// TIA Portal V17 export
// export: Created 2023-05-12T10:40:25.6107869Z, DisplayName Totally Integrated Automation Portal, DisplayVersion V17 Update 4, DisplayName TIA Portal Openness, DisplayVersion V17 Update 4, DisplayName TIA Portal Version Control Interface, DisplayVersion V17, DisplayName STEP 7 Professional, DisplayVersion V17 Update 4, DisplayName STEP 7 Safety, DisplayVersion V17, DisplayName WinCC Advanced / Unified PC, DisplayVersion V17 Update 4
FUNCTION_BLOCK "FB_EM_InputConditioning"   // FB19, LAD
{ S7_Optimized_Access := 'TRUE' }
VERSION : 0.1
// stored: AutoNumber true, CodeModifiedDate 2023-05-12T12:59:41.6492354Z, CompileDate 2023-05-12T12:59:41.6492354Z, CreationDate 2023-05-08T12:19:11.3376827Z, DownloadWithoutReinit false, HandleErrorsWithinBlock false, InterfaceModifiedDate 2023-05-12T12:59:19.7337351Z, IsConsistent true, IsIECCheckEnabled false, IsKnowHowProtected false, IsRetainMemResEnabled false, IsWriteProtected false, LibraryConformanceStatus Warning: The object contains access to global data blocks., MemoryReserve 100, ModifiedDate 2023-05-12T12:59:41.6492354Z, ParameterModified 2022-09-13T10:25:33.4387708Z, PLCSimAdvancedSupport true, SetENOAutomatically false, StructureModified 2023-05-12T12:59:19.7337351Z, UDAEnableTagReadback false
   VAR
      FT01_Przeplyw_Inst { S7_SetPoint := 'True'} : "FB_CM_MeasurementPoint";
      TTs_TempSzafy_Inst { S7_SetPoint := 'True'} : "FB_CM_MeasurementPoint";
      TTz_TempZewn_Inst { S7_SetPoint := 'True'} : "FB_CM_MeasurementPoint";
      PT07_CisnZasil_WRZ6_Inst { S7_SetPoint := 'True'} : "FB_CM_MeasurementPoint";
      PT08_CisnPowr_WRZ6_Inst { S7_SetPoint := 'True'} : "FB_CM_MeasurementPoint";
      TTk_TempKom_Inst { S7_SetPoint := 'True'} : "FB_CM_MeasurementPoint";
      PT01_CisnZasil_PLN1_Inst { S7_SetPoint := 'True'} : "FB_CM_MeasurementPoint";
      PT02_CisnPowr_PLN1_Inst { S7_SetPoint := 'True'} : "FB_CM_MeasurementPoint";
      PT03_CisnZasil_Bypass_Inst { S7_SetPoint := 'True'} : "FB_CM_MeasurementPoint";
      PT04_CisnPowr_Bypass_Inst { S7_SetPoint := 'True'} : "FB_CM_MeasurementPoint";
      PT05_CisnZasil_PLN12_Inst { S7_SetPoint := 'True'} : "FB_CM_MeasurementPoint";
      PT06_CisnPowr_PLN12_Inst { S7_SetPoint := 'True'} : "FB_CM_MeasurementPoint";
      TT01_TempZasil_PLN1_Inst { S7_SetPoint := 'True'} : "FB_CM_MeasurementPoint";
      TT02_TempPowr_PLN1_Inst { S7_SetPoint := 'True'} : "FB_CM_MeasurementPoint";
      TT04_TempPowr_WRZ6_Inst { S7_SetPoint := 'True'} : "FB_CM_MeasurementPoint";
      TT06_TempPowr_PLN12_Inst { S7_SetPoint := 'True'} : "FB_CM_MeasurementPoint";
   END_VAR
BEGIN

REGION Network 1: FT01_Przeplyw - Przepływ
   // FT01_Przeplyw - Przepływ
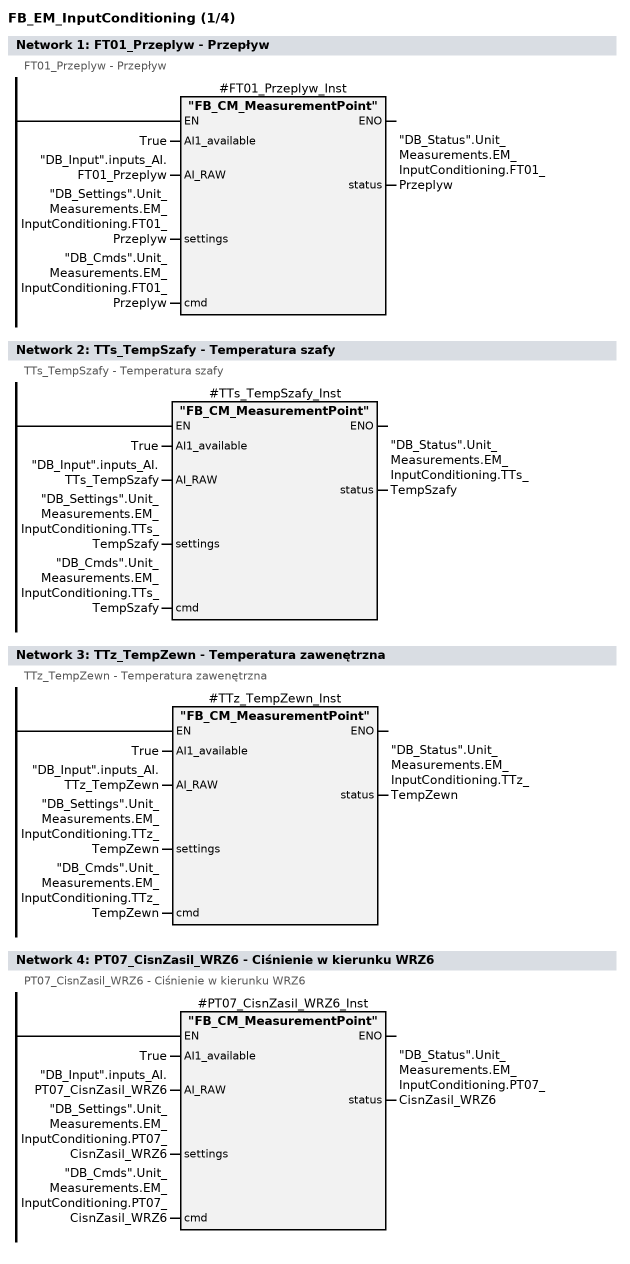
   RUNG wire#powerrail
      #FT01_Przeplyw_Inst(AI1_available := True, AI_RAW := "DB_Input".inputs_AI.FT01_Przeplyw, settings := "DB_Settings".Unit_Measurements.EM_InputConditioning.FT01_Przeplyw, cmd := "DB_Cmds".Unit_Measurements.EM_InputConditioning.FT01_Przeplyw, status => "DB_Status".Unit_Measurements.EM_InputConditioning.FT01_Przeplyw)
   END_RUNG
   // the same network as SCL:
   #FT01_Przeplyw_Inst(AI1_available := True,   // "FB_CM_MeasurementPoint"
                       AI_RAW := "DB_Input".inputs_AI.FT01_Przeplyw,
                       settings := "DB_Settings".Unit_Measurements.EM_InputConditioning.FT01_Przeplyw,
                       cmd := "DB_Cmds".Unit_Measurements.EM_InputConditioning.FT01_Przeplyw,
                       status => "DB_Status".Unit_Measurements.EM_InputConditioning.FT01_Przeplyw);
END_REGION

REGION Network 2: TTs_TempSzafy - Temperatura szafy
   // TTs_TempSzafy - Temperatura szafy
   RUNG wire#powerrail
      #TTs_TempSzafy_Inst(AI1_available := True, AI_RAW := "DB_Input".inputs_AI.TTs_TempSzafy, settings := "DB_Settings".Unit_Measurements.EM_InputConditioning.TTs_TempSzafy, cmd := "DB_Cmds".Unit_Measurements.EM_InputConditioning.TTs_TempSzafy, status => "DB_Status".Unit_Measurements.EM_InputConditioning.TTs_TempSzafy)
   END_RUNG
   // the same network as SCL:
   #TTs_TempSzafy_Inst(AI1_available := True,   // "FB_CM_MeasurementPoint"
                       AI_RAW := "DB_Input".inputs_AI.TTs_TempSzafy,
                       settings := "DB_Settings".Unit_Measurements.EM_InputConditioning.TTs_TempSzafy,
                       cmd := "DB_Cmds".Unit_Measurements.EM_InputConditioning.TTs_TempSzafy,
                       status => "DB_Status".Unit_Measurements.EM_InputConditioning.TTs_TempSzafy);
END_REGION

REGION Network 3: TTz_TempZewn - Temperatura zawenętrzna
   // TTz_TempZewn - Temperatura zawenętrzna
   RUNG wire#powerrail
      #TTz_TempZewn_Inst(AI1_available := True, AI_RAW := "DB_Input".inputs_AI.TTz_TempZewn, settings := "DB_Settings".Unit_Measurements.EM_InputConditioning.TTz_TempZewn, cmd := "DB_Cmds".Unit_Measurements.EM_InputConditioning.TTz_TempZewn, status => "DB_Status".Unit_Measurements.EM_InputConditioning.TTz_TempZewn)
   END_RUNG
   // the same network as SCL:
   #TTz_TempZewn_Inst(AI1_available := True,   // "FB_CM_MeasurementPoint"
                      AI_RAW := "DB_Input".inputs_AI.TTz_TempZewn,
                      settings := "DB_Settings".Unit_Measurements.EM_InputConditioning.TTz_TempZewn,
                      cmd := "DB_Cmds".Unit_Measurements.EM_InputConditioning.TTz_TempZewn,
                      status => "DB_Status".Unit_Measurements.EM_InputConditioning.TTz_TempZewn);
END_REGION

REGION Network 4: PT07_CisnZasil_WRZ6 - Ciśnienie w kierunku WRZ6
   // PT07_CisnZasil_WRZ6 - Ciśnienie w kierunku WRZ6
   RUNG wire#powerrail
      #PT07_CisnZasil_WRZ6_Inst(AI1_available := True, AI_RAW := "DB_Input".inputs_AI.PT07_CisnZasil_WRZ6, settings := "DB_Settings".Unit_Measurements.EM_InputConditioning.PT07_CisnZasil_WRZ6, cmd := "DB_Cmds".Unit_Measurements.EM_InputConditioning.PT07_CisnZasil_WRZ6, status => "DB_Status".Unit_Measurements.EM_InputConditioning.PT07_CisnZasil_WRZ6)
   END_RUNG
   // the same network as SCL:
   #PT07_CisnZasil_WRZ6_Inst(AI1_available := True,   // "FB_CM_MeasurementPoint"
                           AI_RAW := "DB_Input".inputs_AI.PT07_CisnZasil_WRZ6,
                           settings := "DB_Settings".Unit_Measurements.EM_InputConditioning.PT07_CisnZasil_WRZ6,
                           cmd := "DB_Cmds".Unit_Measurements.EM_InputConditioning.PT07_CisnZasil_WRZ6,
                           status => "DB_Status".Unit_Measurements.EM_InputConditioning.PT07_CisnZasil_WRZ6);
END_REGION

REGION Network 5: PT08_CisnPowr_WRZ6 - Ciśnienie powrotu z WRZ6
   // PT08_CisnPowr_WRZ6 - Ciśnienie powrotu z WRZ6
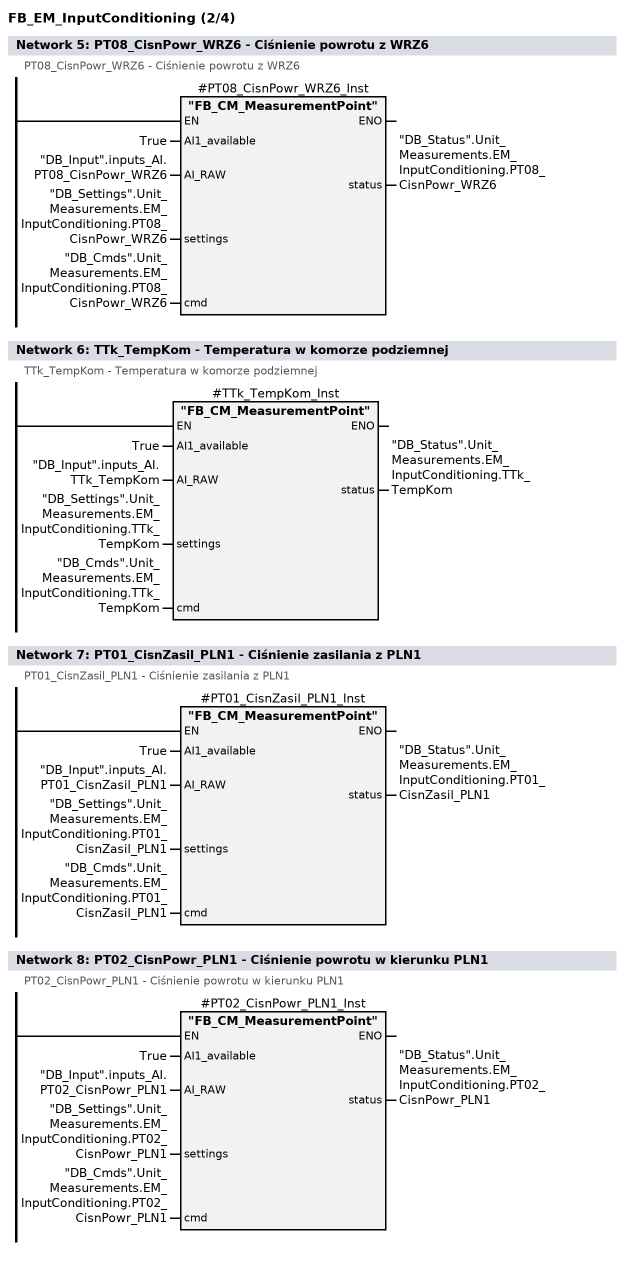
   RUNG wire#powerrail
      #PT08_CisnPowr_WRZ6_Inst(AI1_available := True, AI_RAW := "DB_Input".inputs_AI.PT08_CisnPowr_WRZ6, settings := "DB_Settings".Unit_Measurements.EM_InputConditioning.PT08_CisnPowr_WRZ6, cmd := "DB_Cmds".Unit_Measurements.EM_InputConditioning.PT08_CisnPowr_WRZ6, status => "DB_Status".Unit_Measurements.EM_InputConditioning.PT08_CisnPowr_WRZ6)
   END_RUNG
   // the same network as SCL:
   #PT08_CisnPowr_WRZ6_Inst(AI1_available := True,   // "FB_CM_MeasurementPoint"
                           AI_RAW := "DB_Input".inputs_AI.PT08_CisnPowr_WRZ6,
                           settings := "DB_Settings".Unit_Measurements.EM_InputConditioning.PT08_CisnPowr_WRZ6,
                           cmd := "DB_Cmds".Unit_Measurements.EM_InputConditioning.PT08_CisnPowr_WRZ6,
                           status => "DB_Status".Unit_Measurements.EM_InputConditioning.PT08_CisnPowr_WRZ6);
END_REGION

REGION Network 6: TTk_TempKom - Temperatura w komorze podziemnej
   // TTk_TempKom - Temperatura w komorze podziemnej
   RUNG wire#powerrail
      #TTk_TempKom_Inst(AI1_available := True, AI_RAW := "DB_Input".inputs_AI.TTk_TempKom, settings := "DB_Settings".Unit_Measurements.EM_InputConditioning.TTk_TempKom, cmd := "DB_Cmds".Unit_Measurements.EM_InputConditioning.TTk_TempKom, status => "DB_Status".Unit_Measurements.EM_InputConditioning.TTk_TempKom)
   END_RUNG
   // the same network as SCL:
   #TTk_TempKom_Inst(AI1_available := True,   // "FB_CM_MeasurementPoint"
                     AI_RAW := "DB_Input".inputs_AI.TTk_TempKom,
                     settings := "DB_Settings".Unit_Measurements.EM_InputConditioning.TTk_TempKom,
                     cmd := "DB_Cmds".Unit_Measurements.EM_InputConditioning.TTk_TempKom,
                     status => "DB_Status".Unit_Measurements.EM_InputConditioning.TTk_TempKom);
END_REGION

REGION Network 7: PT01_CisnZasil_PLN1 - Ciśnienie zasilania z PLN1
   // PT01_CisnZasil_PLN1 - Ciśnienie zasilania z PLN1
   RUNG wire#powerrail
      #PT01_CisnZasil_PLN1_Inst(AI1_available := True, AI_RAW := "DB_Input".inputs_AI.PT01_CisnZasil_PLN1, settings := "DB_Settings".Unit_Measurements.EM_InputConditioning.PT01_CisnZasil_PLN1, cmd := "DB_Cmds".Unit_Measurements.EM_InputConditioning.PT01_CisnZasil_PLN1, status => "DB_Status".Unit_Measurements.EM_InputConditioning.PT01_CisnZasil_PLN1)
   END_RUNG
   // the same network as SCL:
   #PT01_CisnZasil_PLN1_Inst(AI1_available := True,   // "FB_CM_MeasurementPoint"
                           AI_RAW := "DB_Input".inputs_AI.PT01_CisnZasil_PLN1,
                           settings := "DB_Settings".Unit_Measurements.EM_InputConditioning.PT01_CisnZasil_PLN1,
                           cmd := "DB_Cmds".Unit_Measurements.EM_InputConditioning.PT01_CisnZasil_PLN1,
                           status => "DB_Status".Unit_Measurements.EM_InputConditioning.PT01_CisnZasil_PLN1);
END_REGION

REGION Network 8: PT02_CisnPowr_PLN1 - Ciśnienie powrotu w kierunku PLN1
   // PT02_CisnPowr_PLN1 - Ciśnienie powrotu w kierunku PLN1
   RUNG wire#powerrail
      #PT02_CisnPowr_PLN1_Inst(AI1_available := True, AI_RAW := "DB_Input".inputs_AI.PT02_CisnPowr_PLN1, settings := "DB_Settings".Unit_Measurements.EM_InputConditioning.PT02_CisnPowr_PLN1, cmd := "DB_Cmds".Unit_Measurements.EM_InputConditioning.PT02_CisnPowr_PLN1, status => "DB_Status".Unit_Measurements.EM_InputConditioning.PT02_CisnPowr_PLN1)
   END_RUNG
   // the same network as SCL:
   #PT02_CisnPowr_PLN1_Inst(AI1_available := True,   // "FB_CM_MeasurementPoint"
                           AI_RAW := "DB_Input".inputs_AI.PT02_CisnPowr_PLN1,
                           settings := "DB_Settings".Unit_Measurements.EM_InputConditioning.PT02_CisnPowr_PLN1,
                           cmd := "DB_Cmds".Unit_Measurements.EM_InputConditioning.PT02_CisnPowr_PLN1,
                           status => "DB_Status".Unit_Measurements.EM_InputConditioning.PT02_CisnPowr_PLN1);
END_REGION

REGION Network 9: PT03_CisnZasil_Bypass - Ciśnienie zasilania Bypass
   // PT03_CisnZasil_Bypass - Ciśnienie zasilania Bypass
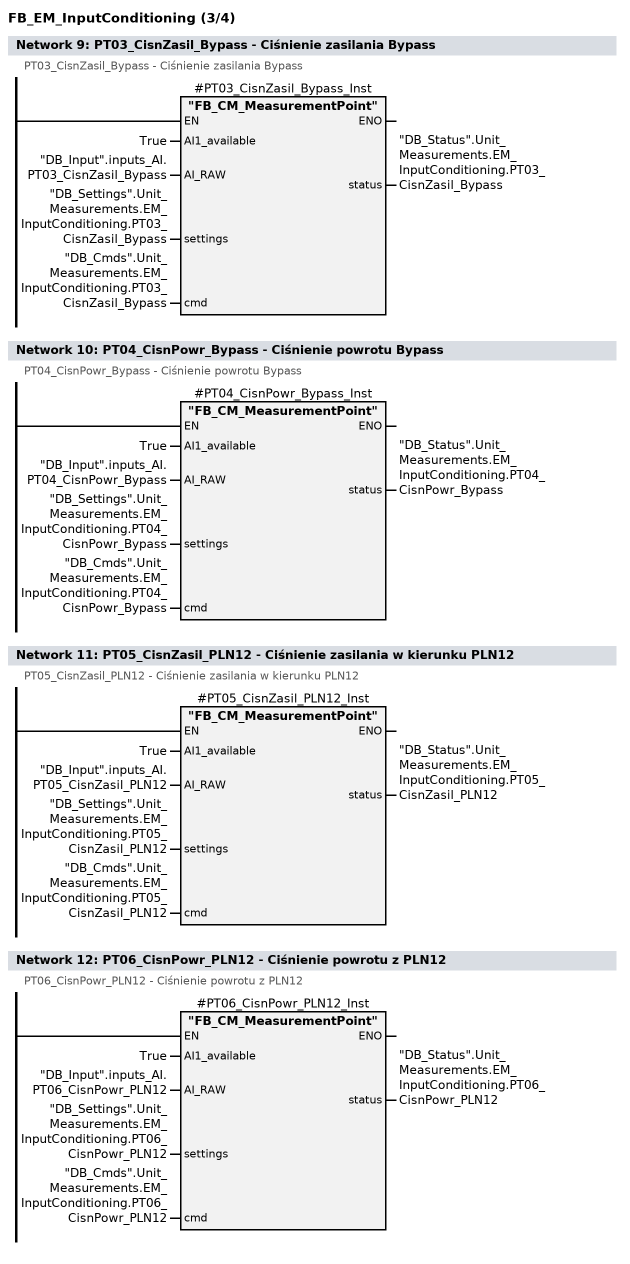
   RUNG wire#powerrail
      #PT03_CisnZasil_Bypass_Inst(AI1_available := True, AI_RAW := "DB_Input".inputs_AI.PT03_CisnZasil_Bypass, settings := "DB_Settings".Unit_Measurements.EM_InputConditioning.PT03_CisnZasil_Bypass, cmd := "DB_Cmds".Unit_Measurements.EM_InputConditioning.PT03_CisnZasil_Bypass, status => "DB_Status".Unit_Measurements.EM_InputConditioning.PT03_CisnZasil_Bypass)
   END_RUNG
   // the same network as SCL:
   #PT03_CisnZasil_Bypass_Inst(AI1_available := True,   // "FB_CM_MeasurementPoint"
                           AI_RAW := "DB_Input".inputs_AI.PT03_CisnZasil_Bypass,
                           settings := "DB_Settings".Unit_Measurements.EM_InputConditioning.PT03_CisnZasil_Bypass,
                           cmd := "DB_Cmds".Unit_Measurements.EM_InputConditioning.PT03_CisnZasil_Bypass,
                           status => "DB_Status".Unit_Measurements.EM_InputConditioning.PT03_CisnZasil_Bypass);
END_REGION

REGION Network 10: PT04_CisnPowr_Bypass - Ciśnienie powrotu Bypass
   // PT04_CisnPowr_Bypass - Ciśnienie powrotu Bypass
   RUNG wire#powerrail
      #PT04_CisnPowr_Bypass_Inst(AI1_available := True, AI_RAW := "DB_Input".inputs_AI.PT04_CisnPowr_Bypass, settings := "DB_Settings".Unit_Measurements.EM_InputConditioning.PT04_CisnPowr_Bypass, cmd := "DB_Cmds".Unit_Measurements.EM_InputConditioning.PT04_CisnPowr_Bypass, status => "DB_Status".Unit_Measurements.EM_InputConditioning.PT04_CisnPowr_Bypass)
   END_RUNG
   // the same network as SCL:
   #PT04_CisnPowr_Bypass_Inst(AI1_available := True,   // "FB_CM_MeasurementPoint"
                           AI_RAW := "DB_Input".inputs_AI.PT04_CisnPowr_Bypass,
                           settings := "DB_Settings".Unit_Measurements.EM_InputConditioning.PT04_CisnPowr_Bypass,
                           cmd := "DB_Cmds".Unit_Measurements.EM_InputConditioning.PT04_CisnPowr_Bypass,
                           status => "DB_Status".Unit_Measurements.EM_InputConditioning.PT04_CisnPowr_Bypass);
END_REGION

REGION Network 11: PT05_CisnZasil_PLN12 - Ciśnienie zasilania w kierunku PLN12
   // PT05_CisnZasil_PLN12 - Ciśnienie zasilania w kierunku PLN12
   RUNG wire#powerrail
      #PT05_CisnZasil_PLN12_Inst(AI1_available := True, AI_RAW := "DB_Input".inputs_AI.PT05_CisnZasil_PLN12, settings := "DB_Settings".Unit_Measurements.EM_InputConditioning.PT05_CisnZasil_PLN12, cmd := "DB_Cmds".Unit_Measurements.EM_InputConditioning.PT05_CisnZasil_PLN12, status => "DB_Status".Unit_Measurements.EM_InputConditioning.PT05_CisnZasil_PLN12)
   END_RUNG
   // the same network as SCL:
   #PT05_CisnZasil_PLN12_Inst(AI1_available := True,   // "FB_CM_MeasurementPoint"
                           AI_RAW := "DB_Input".inputs_AI.PT05_CisnZasil_PLN12,
                           settings := "DB_Settings".Unit_Measurements.EM_InputConditioning.PT05_CisnZasil_PLN12,
                           cmd := "DB_Cmds".Unit_Measurements.EM_InputConditioning.PT05_CisnZasil_PLN12,
                           status => "DB_Status".Unit_Measurements.EM_InputConditioning.PT05_CisnZasil_PLN12);
END_REGION

REGION Network 12: PT06_CisnPowr_PLN12 - Ciśnienie powrotu z PLN12
   // PT06_CisnPowr_PLN12 - Ciśnienie powrotu z PLN12
   RUNG wire#powerrail
      #PT06_CisnPowr_PLN12_Inst(AI1_available := True, AI_RAW := "DB_Input".inputs_AI.PT06_CisnPowr_PLN12, settings := "DB_Settings".Unit_Measurements.EM_InputConditioning.PT06_CisnPowr_PLN12, cmd := "DB_Cmds".Unit_Measurements.EM_InputConditioning.PT06_CisnPowr_PLN12, status => "DB_Status".Unit_Measurements.EM_InputConditioning.PT06_CisnPowr_PLN12)
   END_RUNG
   // the same network as SCL:
   #PT06_CisnPowr_PLN12_Inst(AI1_available := True,   // "FB_CM_MeasurementPoint"
                           AI_RAW := "DB_Input".inputs_AI.PT06_CisnPowr_PLN12,
                           settings := "DB_Settings".Unit_Measurements.EM_InputConditioning.PT06_CisnPowr_PLN12,
                           cmd := "DB_Cmds".Unit_Measurements.EM_InputConditioning.PT06_CisnPowr_PLN12,
                           status => "DB_Status".Unit_Measurements.EM_InputConditioning.PT06_CisnPowr_PLN12);
END_REGION

REGION Network 13: TT01_TempZasil_PLN1 - Temperatura zasliania z PLN1
   // TT01_TempZasil_PLN1 - Temperatura zasliania z PLN1
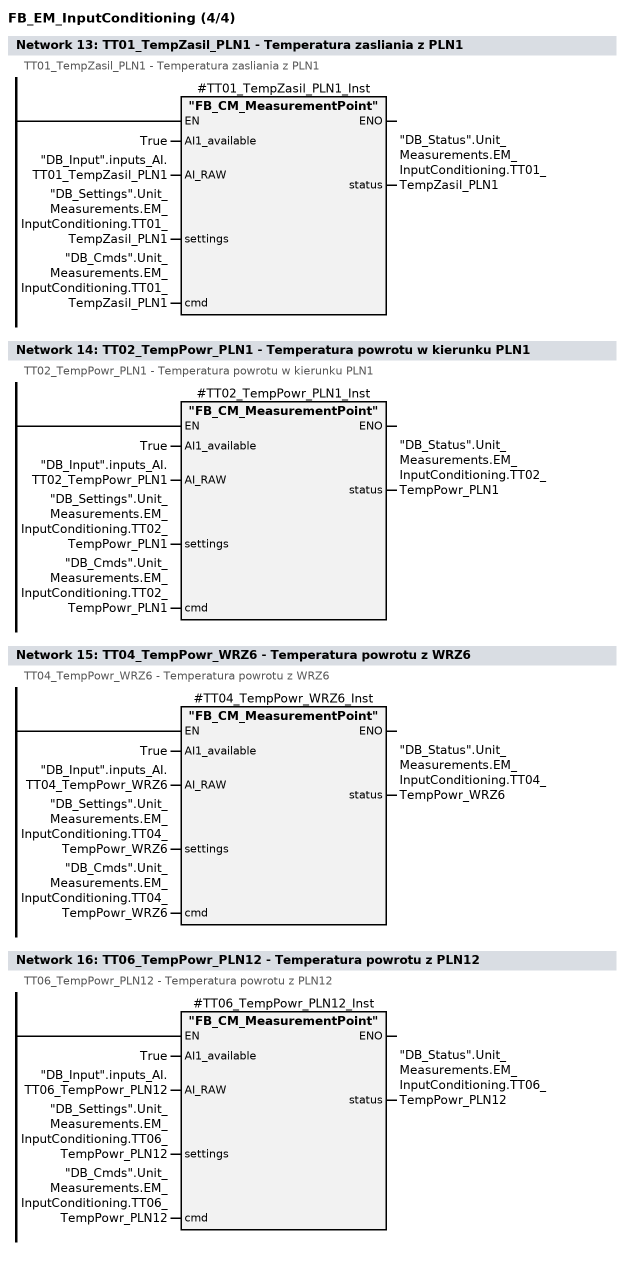
   RUNG wire#powerrail
      #TT01_TempZasil_PLN1_Inst(AI1_available := True, AI_RAW := "DB_Input".inputs_AI.TT01_TempZasil_PLN1, settings := "DB_Settings".Unit_Measurements.EM_InputConditioning.TT01_TempZasil_PLN1, cmd := "DB_Cmds".Unit_Measurements.EM_InputConditioning.TT01_TempZasil_PLN1, status => "DB_Status".Unit_Measurements.EM_InputConditioning.TT01_TempZasil_PLN1)
   END_RUNG
   // the same network as SCL:
   #TT01_TempZasil_PLN1_Inst(AI1_available := True,   // "FB_CM_MeasurementPoint"
                           AI_RAW := "DB_Input".inputs_AI.TT01_TempZasil_PLN1,
                           settings := "DB_Settings".Unit_Measurements.EM_InputConditioning.TT01_TempZasil_PLN1,
                           cmd := "DB_Cmds".Unit_Measurements.EM_InputConditioning.TT01_TempZasil_PLN1,
                           status => "DB_Status".Unit_Measurements.EM_InputConditioning.TT01_TempZasil_PLN1);
END_REGION

REGION Network 14: TT02_TempPowr_PLN1 - Temperatura powrotu w kierunku PLN1
   // TT02_TempPowr_PLN1 - Temperatura powrotu w kierunku PLN1
   RUNG wire#powerrail
      #TT02_TempPowr_PLN1_Inst(AI1_available := True, AI_RAW := "DB_Input".inputs_AI.TT02_TempPowr_PLN1, settings := "DB_Settings".Unit_Measurements.EM_InputConditioning.TT02_TempPowr_PLN1, cmd := "DB_Cmds".Unit_Measurements.EM_InputConditioning.TT02_TempPowr_PLN1, status => "DB_Status".Unit_Measurements.EM_InputConditioning.TT02_TempPowr_PLN1)
   END_RUNG
   // the same network as SCL:
   #TT02_TempPowr_PLN1_Inst(AI1_available := True,   // "FB_CM_MeasurementPoint"
                           AI_RAW := "DB_Input".inputs_AI.TT02_TempPowr_PLN1,
                           settings := "DB_Settings".Unit_Measurements.EM_InputConditioning.TT02_TempPowr_PLN1,
                           cmd := "DB_Cmds".Unit_Measurements.EM_InputConditioning.TT02_TempPowr_PLN1,
                           status => "DB_Status".Unit_Measurements.EM_InputConditioning.TT02_TempPowr_PLN1);
END_REGION

REGION Network 15: TT04_TempPowr_WRZ6 - Temperatura powrotu z WRZ6
   // TT04_TempPowr_WRZ6 - Temperatura powrotu z WRZ6
   RUNG wire#powerrail
      #TT04_TempPowr_WRZ6_Inst(AI1_available := True, AI_RAW := "DB_Input".inputs_AI.TT04_TempPowr_WRZ6, settings := "DB_Settings".Unit_Measurements.EM_InputConditioning.TT04_TempPowr_WRZ6, cmd := "DB_Cmds".Unit_Measurements.EM_InputConditioning.TT04_TempPowr_WRZ6, status => "DB_Status".Unit_Measurements.EM_InputConditioning.TT04_TempPowr_WRZ6)
   END_RUNG
   // the same network as SCL:
   #TT04_TempPowr_WRZ6_Inst(AI1_available := True,   // "FB_CM_MeasurementPoint"
                           AI_RAW := "DB_Input".inputs_AI.TT04_TempPowr_WRZ6,
                           settings := "DB_Settings".Unit_Measurements.EM_InputConditioning.TT04_TempPowr_WRZ6,
                           cmd := "DB_Cmds".Unit_Measurements.EM_InputConditioning.TT04_TempPowr_WRZ6,
                           status => "DB_Status".Unit_Measurements.EM_InputConditioning.TT04_TempPowr_WRZ6);
END_REGION

REGION Network 16: TT06_TempPowr_PLN12 - Temperatura powrotu z PLN12
   // TT06_TempPowr_PLN12 - Temperatura powrotu z PLN12
   RUNG wire#powerrail
      #TT06_TempPowr_PLN12_Inst(AI1_available := True, AI_RAW := "DB_Input".inputs_AI.TT06_TempPowr_PLN12, settings := "DB_Settings".Unit_Measurements.EM_InputConditioning.TT06_TempPowr_PLN12, cmd := "DB_Cmds".Unit_Measurements.EM_InputConditioning.TT06_TempPowr_PLN12, status => "DB_Status".Unit_Measurements.EM_InputConditioning.TT06_TempPowr_PLN12)
   END_RUNG
   // the same network as SCL:
   #TT06_TempPowr_PLN12_Inst(AI1_available := True,   // "FB_CM_MeasurementPoint"
                           AI_RAW := "DB_Input".inputs_AI.TT06_TempPowr_PLN12,
                           settings := "DB_Settings".Unit_Measurements.EM_InputConditioning.TT06_TempPowr_PLN12,
                           cmd := "DB_Cmds".Unit_Measurements.EM_InputConditioning.TT06_TempPowr_PLN12,
                           status => "DB_Status".Unit_Measurements.EM_InputConditioning.TT06_TempPowr_PLN12);
END_REGION
END_FUNCTION_BLOCK
